Staubli VAL3: recvMsgBody.pgx

public program recvMsgBody(num& x_nMsgRecvState (dimensions=1))
  local bool l_bFlag
begin
  // Copyright (c) 2016, Ocado Technology - Robotics Research Team
  //
  // Licensed under the Apache License, Version 2.0 (the "License");
  // you may not use this file except in compliance with the License.
  // You may obtain a copy of the License at
  //
  //     http://www.apache.org/licenses/LICENSE-2.0
  //
  // Unless required by applicable law or agreed to in writing, software
  // distributed under the License is distributed on an "AS IS" BASIS,
  // WITHOUT WARRANTIES OR CONDITIONS OF ANY KIND, either express or implied.
  // See the License for the specific language governing permissions and
  // limitations under the License.



  l_bFlag=false

  switch rosGenericMsg.header.nMsgType
    case 11
      call recvTrajPt(l_bFlag)
    break
    case 14
      call recvTrajPtFull(l_bFlag)
    break
    default
    break
  endSwitch

  if (l_bFlag==true)
    // move on to state 3: decode msg body
    x_nMsgRecvState=3
  else
    // error whilst receiving msg body, reset state machine
    x_nMsgRecvState=0
  endIf
end
